# EPICS substitutions: daq6510/Db/daq6510.substitutions
file "daq6510-gen.template" { pattern
{}
{}
}

file "daq6510-chan.template" { pattern
{CHAN}
{01}
{02}
{03}
{04}
{05}
{06}
{07}
{08}
{09}
{10}
{11}
{12}
{13}
{14}
{15}
{16}
{17}
{18}
{19}
{20}
}
